PROGRAM Control_Panel_FSM
VAR
END_VAR

END_PROGRAM

(* stored: Version 1.1.0.1, ProductVersion 3.1.4024.15
   POU Control_Panel_FSM: Id {25b0d9bf-0951-41c2-af0f-f76219c646b4}, SpecialFunc None *)
